FUNCTION ASSEMBLE_DWORD_FROM_WORDS (* this Function combines the 2 WORDS to a dword *)
  (* Standard: 61499-1; Description: Copyright (c) 2024 HR Agrartechnik GmbH This program and the accompanying materials are made available under the terms of the Eclipse Public License 2.0 which is available at https://www.eclipse.org/legal/epl-2.0/ SPDX-License-Identifier: EPL-2.0 *)
  (* Version 3.0, 2025-04-14, Patrick Aigner, changed package *)
  (* Version 1.1, 2024-07-28, Moritz Ortmeier, HR Agrartechnik, rename Function and change Input/Output Variables *)
  (* Version 1.0, 2024-02-22, Franz Höpfinger, HR Agrartechnik, initial Implementation *)
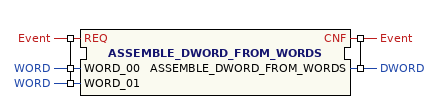
  EVENT_INPUT
    REQ WITH WORD_00, WORD_01;
  END_EVENT
  EVENT_OUTPUT
    CNF WITH ASSEMBLE_DWORD_FROM_WORDS;
  END_EVENT
  VAR_INPUT
    WORD_00 : WORD;
    WORD_01 : WORD;
  END_VAR
  VAR_OUTPUT
    ASSEMBLE_DWORD_FROM_WORDS : DWORD;
  END_VAR
  BODY IN ST:
(* this Function combines the 2 WORDS to a dword *)
FUNCTION ASSEMBLE_DWORD_FROM_WORDS : DWORD

VAR_INPUT
	WORD_00 : WORD;
	WORD_01 : WORD;
END_VAR

ASSEMBLE_DWORD_FROM_WORDS.%W0 := WORD_00;
ASSEMBLE_DWORD_FROM_WORDS.%W1 := WORD_01;

END_FUNCTION
  END_BODY
END_FUNCTION
